FUNCTION_BLOCK RSFlipFlop
VAR_INPUT											//S-Dominanter RS-Baustein
	bSET: BOOL;										//Baustein-interne Set-Variable
	bRESET: BOOL;									//Baustein-interne Reset-Variable
END_VAR
VAR_OUTPUT
END_VAR
VAR
	RSFlipFlop: RS;									//Instanziierung des RS-Bausteins
END_VAR

RSFlipFlop(SET:= bSET, RESET1:= bRESET);			//Verknüpfung der Baustein-internen Variablen mit den Bausteineingängen

END_FUNCTION_BLOCK

(* stored: Version 1.1.0.1
   POU RSFlipFlop: Id {2a7bc940-8e73-43ad-ac5e-48a14135cb88}, SpecialFunc None *)
